{attribute 'GeneratedUsingTerminal: EL9930-0000-0016'}
{attribute addProperty BoxType "EL9930-0000-0016"}
{attribute addProperty Id "EtcSlaveTerminalBaseIO_InputsEMPTY_STRUCTURE0IO_OutputsEMPTY_STRUCTURE0WcStateAT %I*WcState_9091E0EB2InfoDataAT %I*InfoData_90184F0C16"}
{attribute addProperty CRC "3819992516"}
{attribute addProperty Size "18"}
TYPE EL9930_E3B075C4 EXTENDS EtcSlaveTerminalBase :
STRUCT
	{attribute addProperty Name "IO_Inputs"}
	IO_Inputs : EMPTY_STRUCTURE;
	{attribute addProperty Name "IO_Outputs"}
	IO_Outputs : EMPTY_STRUCTURE;
	{attribute addProperty Name "WcState"}
	WcState : WcState_9091E0EB;
	{attribute addProperty Name "InfoData"}
	InfoData : InfoData_90184F0C;
END_STRUCT
END_TYPE

(* stored: Version 1.2.0.0, ProductVersion 3.1.4024.9
   DUT EL9930_E3B075C4: Id {18396e03-8462-4dbe-9ff5-5bf0f4b3ab78} *)
